KUKA KRL program: dai_before_zero.src, dai_before_zero.dat

--- dai_before_zero.src ---
&ACCESS RVP
&COMMENT dai_robot_check
&USER thsc160
&PARAM version = 0.1
DEF dai_before_zero( )
;FOLD INI
  ;FOLD BASISTECH INI
    GLOBAL INTERRUPT DECL 3 WHEN $STOPMESS==TRUE DO IR_STOPM ( )
    BAS (#INITMOV,0 )
  ;ENDFOLD (BASISTECH INI)
;FOLD SPOTTECH INI
USERSPOT(#INIT)
;ENDFOLD (SPOTTECH INI)
;FOLD GRIPPERTECH INI
USER_GRP(0,DUMMY,DUMMY,GDEFAULT)
;ENDFOLD (GRIPPERTECH INI)
;FOLD USER INI

;Make your modifications here
;FOLD COLLISION_V_3.01 INI ;%{E}
    IF (COLLISION_DATA[1].I_NR>0) THEN
    GLOBAL INTERRUPT DECL 21 WHEN $IN[COLLISION_DATA[1].I_NR]==FALSE DO COLLSTOP (1,0 )
    ENDIF
    IF (COLLISION_DATA[2].I_NR>0) THEN
    GLOBAL INTERRUPT DECL 22 WHEN $IN[COLLISION_DATA[2].I_NR]==FALSE DO COLLSTOP (2,0 )
    ENDIF
    IF (COLLISION_DATA[3].I_NR>0) THEN
    GLOBAL INTERRUPT DECL 23 WHEN $IN[COLLISION_DATA[3].I_NR]==FALSE DO COLLSTOP (3,0 )
    ENDIF
    IF (COLLISION_DATA[4].I_NR>0) THEN
    GLOBAL INTERRUPT DECL 24 WHEN $IN[COLLISION_DATA[4].I_NR]==FALSE DO COLLSTOP (4,0 )
    ENDIF
;ENDFOLD (Collision)

;ENDFOLD (USER INI)

;ENDFOLD (INI)

;FOLD ; machine identifier:;%{PE}%R 8.2.11,%MKUKATPBASIS,%CCOMMENT,%VNORMAL,%P 2:machine identifier:
;ENDFOLD
;FOLD ; station-nr.:;%{PE}%R 5.4.33,%MKUKATPBASIS,%CCOMMENT,%VNORMAL,%P 2:station-nr.:
;ENDFOLD
;FOLD ; version:;%{PE}%R 8.2.11,%MKUKATPBASIS,%CCOMMENT,%VNORMAL,%P 2:version:
;ENDFOLD
;FOLD ; name arranger:;%{PE}%R 5.4.33,%MKUKATPBASIS,%CCOMMENT,%VNORMAL,%P 2:name arranger:
;ENDFOLD


;only in template, remove after teaching
wait for false


REPEAT
  MSG_SHOW("H_Prog",#quit,999,"dai_rob_ok_0")
UNTIL $T1 == TRUE

; ***************************************
; A T T E N T I O N !!! Only drive in $T1
; ***************************************

;FOLD PTP HOME Vel=100 % DEFAULT;%{PE}%R 5.5.24,%MKUKATPBASIS,%CMOVE,%VPTP,%P 1:PTP, 2:HOME, 3:, 5:100, 7:DEFAULT
$BWDSTART=FALSE
PDAT_ACT=PDEFAULT
FDAT_ACT=FHOME
BAS(#PTP_PARAMS,100)
$H_POS=XHOME
PTP XHOME
;ENDFOLD


MSG_SHOW("H_Prog",#dialog,1,"dai_before_zero_1")
WHILE TRUE
;zum Anfahren der Nullstellung Satzzeiger setzen
;for approaching the zero set record pointer
HALT
ENDWHILE

; teach the way to Mech-Zero
;FOLD PTP LHP1  Vel= 100 % PDEFAULT Tool[64] Base[64];%{PE}%R 5.2.7,%MKUKATPBASIS,%CMOVE,%VPTP,%P 1:PTP, 2:LHP1, 3:, 5:100, 7:PDEFAULT
    $BWDSTART = FALSE
    PDAT_ACT=PPDEFAULT
    FDAT_ACT=FLHP1
    BAS(#PTP_PARAMS,100)
    PTP XLHP1
;ENDFOLD
;FOLD PTP LHP2  Vel= 100 % PDEFAULT Tool[64] Base[64];%{PE}%R 5.2.7,%MKUKATPBASIS,%CMOVE,%VPTP,%P 1:PTP, 2:LHP2, 3:, 5:100, 7:PDEFAULT
    $BWDSTART = FALSE
    PDAT_ACT=PPDEFAULT
    FDAT_ACT=FLHP2
    BAS(#PTP_PARAMS,100)
    PTP XLHP2
;ENDFOLD

;FOLD ; Mechanische Null | mechanical zero;%{PE}%R 3.2.24,%MKUKATPBASIS,%CCOMMENT,%VNORMAL,%P 2:Mechanische Null | mechanical zero
;ENDFOLD
MSG_SHOW("H_Prog",#dialog,2,"dai_before_zero_2")

;FOLD PTP Mechnull  Vel= 100 % PDEFAULT;%{PE}%R 3.2.24,%MKUKATPBASIS,%CMOVE,%VPTP,%P 1:PTP, 2:Mechnull, 3:, 5:100, 7:PDEFAULT
    $BWDSTART = FALSE
    PDAT_ACT=PPDEFAULT
    BAS(#PTP_DAT)
    FDAT_ACT=FMechnull
    BAS(#FRAMES)
    BAS(#VEL_PTP,100)
    PTP XMechnull
;ENDFOLD
HALT

;FOLD ; Kerben anfahren | Approach scores ;%{PE}%R 3.2.24,%MKUKATPBASIS,%CCOMMENT,%VNORMAL,%P 2:Kerben anfahren | Approach scores
;ENDFOLD
MSG_SHOW("H_Prog",#dialog,3,"dai_before_zero_3")
;FOLD PTP Vorjus  Vel= 100 % PDEFAULT;%{PE}%R 3.2.24,%MKUKATPBASIS,%CMOVE,%VPTP,%P 1:PTP, 2:Vorjus, 3:, 5:100, 7:PDEFAULT
    $BWDSTART = FALSE
    PDAT_ACT=PPDEFAULT
    BAS(#PTP_DAT)
    FDAT_ACT=FVorjus
    BAS(#FRAMES)
    BAS(#VEL_PTP,100)
    PTP XVorjus
;ENDFOLD

;FOLD ; ------------------------------;%{PE}%R 3.2.24,%MKUKATPBASIS,%CCOMMENT,%VNORMAL,%P 2:------------------------------
;ENDFOLD
;FOLD ; Justage! | Calibration;%{PE}%R 3.2.24,%MKUKATPBASIS,%CCOMMENT,%VNORMAL,%P 2: Justage! | Calibration
;ENDFOLD
;FOLD ; ------------------------------;%{PE}%R 3.2.24,%MKUKATPBASIS,%CCOMMENT,%VNORMAL,%P 2:------------------------------
;ENDFOLD
;FOLD ; Nullstellung mit Werkzeug | Zero-Position with tool ;%{PE}%R 3.2.24,%MKUKATPBASIS,%CCOMMENT,%VNORMAL,%P 2:Nullstellung mit Werkzeug | Zero-Position with tool
;ENDFOLD

MSG_SHOW("H_Prog",#dialog,4,"dai_before_zero_4")



;FOLD PTP HOME Vel=100 % DEFAULT;%{PE}%R 5.5.24,%MKUKATPBASIS,%CMOVE,%VPTP,%P 1:PTP, 2:HOME, 3:, 5:100, 7:DEFAULT
$BWDSTART=FALSE
PDAT_ACT=PDEFAULT
FDAT_ACT=FHOME
BAS(#PTP_PARAMS,100)
$H_POS=XHOME
PTP XHOME
;ENDFOLD

END

--- dai_before_zero.dat ---
&ACCESS RVP
&COMMENT dai_robot_check
&USER thsc160
&PARAM version = 0.1
DEFDAT dai_before_zero
;FOLD EXTERNAL DECLARATIONS;%{PE}%MKUKATPBASIS,%CEXT,%VCOMMON,%P
;FOLD GRIPPERTECH EXT
  EXT  H50 (INT:IN, INT:IN ,INT:IN ,GRP_TYP:IN)
;ENDFOLD (GRIPPERTECH EXT)
;FOLD SPOTTECH EXT
  EXT  USERSPOT (S_COMMAND  :IN, SPOT_TYPE:IN)
;ENDFOLD (SPOTTECH EXT)
;FOLD BASISTECH EXT;%{PE}%MKUKATPBASIS,%CEXT,%VEXT,%P
EXT  BAS (BAS_COMMAND  :IN,REAL  :IN )
DECL INT SUCCESS
;ENDFOLD (BASISTECH EXT)
;FOLD USER EXT;%{E}%MKUKATPUSER,%CEXT,%VEXT,%P
;Make here your modifications
;FOLD COLLISION
EXT  COLLSTOP (INT  :IN,INT  :IN )
;ENDFOLD  (Collision)
;ENDFOLD (USER EXT)
;ENDFOLD (EXTERNAL DECLERATIONS)

DECL BASIS_SUGG_T LAST_BASIS={POINT1[] "P0                      ",POINT2[] "P0                      ",CP_PARAMS[] "CPDAT0                  ",PTP_PARAMS[] "PDAT0                  ",CONT[] "                        ",CP_VEL[] "2                       ",PTP_VEL[] "100                     "}

E6AXIS XVORJUS={A1 0.699999988,A2 -89.0,A3 91.1999969,A4 6.0,A5 2.5,A6 4.0,E1 0.0,E2 0.0,E3 0.0,E4 0.0,E5 0.0,E6 0.0}
DECL E6POS XLHP1={X 0.0,Y 0.0,Z 0.0,A 0.0,B 0.0,C 0.0,S 2,T 2,E1 0.0,E2 0.0,E3 0.0,E4 0.0,E5 0.0,E6 0.0}
DECL E6POS XLHP2={X 0.0,Y 0.0,Z 0.0,A 0.0,B 0.0,C 0.0,S 2,T 2,E1 0.0,E2 0.0,E3 0.0,E4 0.0,E5 0.0,E6 0.0}
DECL PDAT PPDEFAULT={VEL 100.0,ACC 100.0,APO_DIST 100.0}
DECL FDAT FVORJUS={TOOL_NO 64,BASE_NO 64,IPO_FRAME #BASE}
DECL FDAT FLHP1={TOOL_NO 64,BASE_NO 64,IPO_FRAME #BASE,POINT2[] " "}
DECL FDAT FLHP2={TOOL_NO 64,BASE_NO 64,IPO_FRAME #BASE,POINT2[] " "}
DECL FDAT FHOME={TOOL_NO 64,BASE_NO 64,IPO_FRAME #BASE,POINT2[] " "}
DECL FDAT FCONTROLL1={TOOL_NO 16,BASE_NO 16,IPO_FRAME #BASE,POINT2[] " ",TQ_STATE FALSE}

ENDDAT
